{attribute addProperty BoxType "KL6211-0002"}
{attribute addProperty Id "Channel_1Channel_E3914DFD00"}
{attribute addProperty CRC "1423467616"}
{attribute addProperty SizeInBites "0"}
{attribute addProperty SizeInBytes "0"}
TYPE KL_54D86460 :
STRUCT
	{attribute addProperty Name "Channel_1"}
	Channel_1 : Channel_E3914DFD;
END_STRUCT
END_TYPE

(* stored: Version 1.2.0.0, ProductVersion 3.1.4024.9
   DUT KL_54D86460: Id {3e6347b6-be7b-42c4-8532-c0590ed37fb2} *)
